REGION Network 11: Extrusora 11
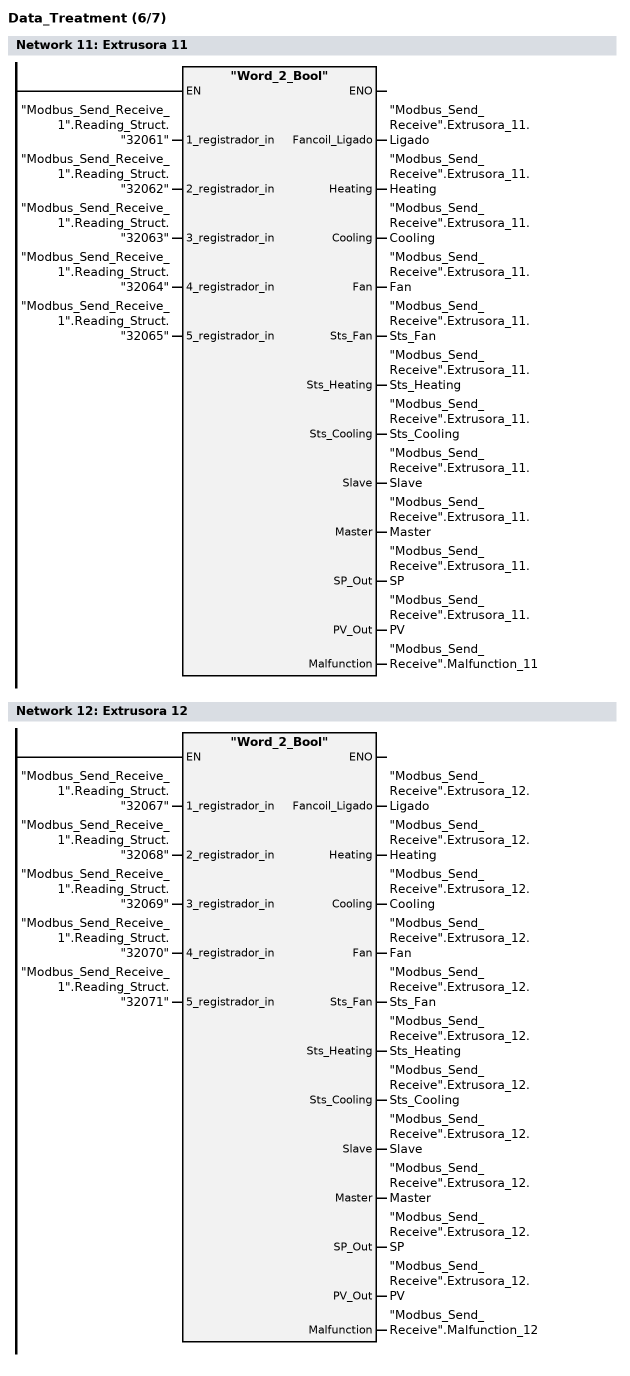
   RUNG wire#powerrail
      "Word_2_Bool"("1_registrador_in" := "Modbus_Send_Receive_1".Reading_Struct."32061", "2_registrador_in" := "Modbus_Send_Receive_1".Reading_Struct."32062", "3_registrador_in" := "Modbus_Send_Receive_1".Reading_Struct."32063", "4_registrador_in" := "Modbus_Send_Receive_1".Reading_Struct."32064", "5_registrador_in" := "Modbus_Send_Receive_1".Reading_Struct."32065", Fancoil_Ligado => "Modbus_Send_Receive".Extrusora_11.Ligado, Heating => "Modbus_Send_Receive".Extrusora_11.Heating, Cooling => "Modbus_Send_Receive".Extrusora_11.Cooling, Fan => "Modbus_Send_Receive".Extrusora_11.Fan, Sts_Fan => "Modbus_Send_Receive".Extrusora_11.Sts_Fan, Sts_Heating => "Modbus_Send_Receive".Extrusora_11.Sts_Heating, Sts_Cooling => "Modbus_Send_Receive".Extrusora_11.Sts_Cooling, Slave => "Modbus_Send_Receive".Extrusora_11.Slave, Master => "Modbus_Send_Receive".Extrusora_11.Master, SP_Out => "Modbus_Send_Receive".Extrusora_11.SP, PV_Out => "Modbus_Send_Receive".Extrusora_11.PV, Malfunction => "Modbus_Send_Receive".Malfunction_11)
   END_RUNG
   // the same network as SCL:
   "Word_2_Bool"("1_registrador_in" := "Modbus_Send_Receive_1".Reading_Struct."32061",
                 "2_registrador_in" := "Modbus_Send_Receive_1".Reading_Struct."32062",
                 "3_registrador_in" := "Modbus_Send_Receive_1".Reading_Struct."32063",
                 "4_registrador_in" := "Modbus_Send_Receive_1".Reading_Struct."32064",
                 "5_registrador_in" := "Modbus_Send_Receive_1".Reading_Struct."32065",
                 Fancoil_Ligado => "Modbus_Send_Receive".Extrusora_11.Ligado,
                 Heating => "Modbus_Send_Receive".Extrusora_11.Heating,
                 Cooling => "Modbus_Send_Receive".Extrusora_11.Cooling,
                 Fan => "Modbus_Send_Receive".Extrusora_11.Fan,
                 Sts_Fan => "Modbus_Send_Receive".Extrusora_11.Sts_Fan,
                 Sts_Heating => "Modbus_Send_Receive".Extrusora_11.Sts_Heating,
                 Sts_Cooling => "Modbus_Send_Receive".Extrusora_11.Sts_Cooling,
                 Slave => "Modbus_Send_Receive".Extrusora_11.Slave,
                 Master => "Modbus_Send_Receive".Extrusora_11.Master,
                 SP_Out => "Modbus_Send_Receive".Extrusora_11.SP,
                 PV_Out => "Modbus_Send_Receive".Extrusora_11.PV,
                 Malfunction => "Modbus_Send_Receive".Malfunction_11);
END_REGION

REGION Network 12: Extrusora 12
   RUNG wire#powerrail
      "Word_2_Bool"("1_registrador_in" := "Modbus_Send_Receive_1".Reading_Struct."32067", "2_registrador_in" := "Modbus_Send_Receive_1".Reading_Struct."32068", "3_registrador_in" := "Modbus_Send_Receive_1".Reading_Struct."32069", "4_registrador_in" := "Modbus_Send_Receive_1".Reading_Struct."32070", "5_registrador_in" := "Modbus_Send_Receive_1".Reading_Struct."32071", Fancoil_Ligado => "Modbus_Send_Receive".Extrusora_12.Ligado, Heating => "Modbus_Send_Receive".Extrusora_12.Heating, Cooling => "Modbus_Send_Receive".Extrusora_12.Cooling, Fan => "Modbus_Send_Receive".Extrusora_12.Fan, Sts_Fan => "Modbus_Send_Receive".Extrusora_12.Sts_Fan, Sts_Heating => "Modbus_Send_Receive".Extrusora_12.Sts_Heating, Sts_Cooling => "Modbus_Send_Receive".Extrusora_12.Sts_Cooling, Slave => "Modbus_Send_Receive".Extrusora_12.Slave, Master => "Modbus_Send_Receive".Extrusora_12.Master, SP_Out => "Modbus_Send_Receive".Extrusora_12.SP, PV_Out => "Modbus_Send_Receive".Extrusora_12.PV, Malfunction => "Modbus_Send_Receive".Malfunction_12)
   END_RUNG
   // the same network as SCL:
   "Word_2_Bool"("1_registrador_in" := "Modbus_Send_Receive_1".Reading_Struct."32067",
                 "2_registrador_in" := "Modbus_Send_Receive_1".Reading_Struct."32068",
                 "3_registrador_in" := "Modbus_Send_Receive_1".Reading_Struct."32069",
                 "4_registrador_in" := "Modbus_Send_Receive_1".Reading_Struct."32070",
                 "5_registrador_in" := "Modbus_Send_Receive_1".Reading_Struct."32071",
                 Fancoil_Ligado => "Modbus_Send_Receive".Extrusora_12.Ligado,
                 Heating => "Modbus_Send_Receive".Extrusora_12.Heating,
                 Cooling => "Modbus_Send_Receive".Extrusora_12.Cooling,
                 Fan => "Modbus_Send_Receive".Extrusora_12.Fan,
                 Sts_Fan => "Modbus_Send_Receive".Extrusora_12.Sts_Fan,
                 Sts_Heating => "Modbus_Send_Receive".Extrusora_12.Sts_Heating,
                 Sts_Cooling => "Modbus_Send_Receive".Extrusora_12.Sts_Cooling,
                 Slave => "Modbus_Send_Receive".Extrusora_12.Slave,
                 Master => "Modbus_Send_Receive".Extrusora_12.Master,
                 SP_Out => "Modbus_Send_Receive".Extrusora_12.SP,
                 PV_Out => "Modbus_Send_Receive".Extrusora_12.PV,
                 Malfunction => "Modbus_Send_Receive".Malfunction_12);
END_REGION

REGION Network 13: Extrusora 13
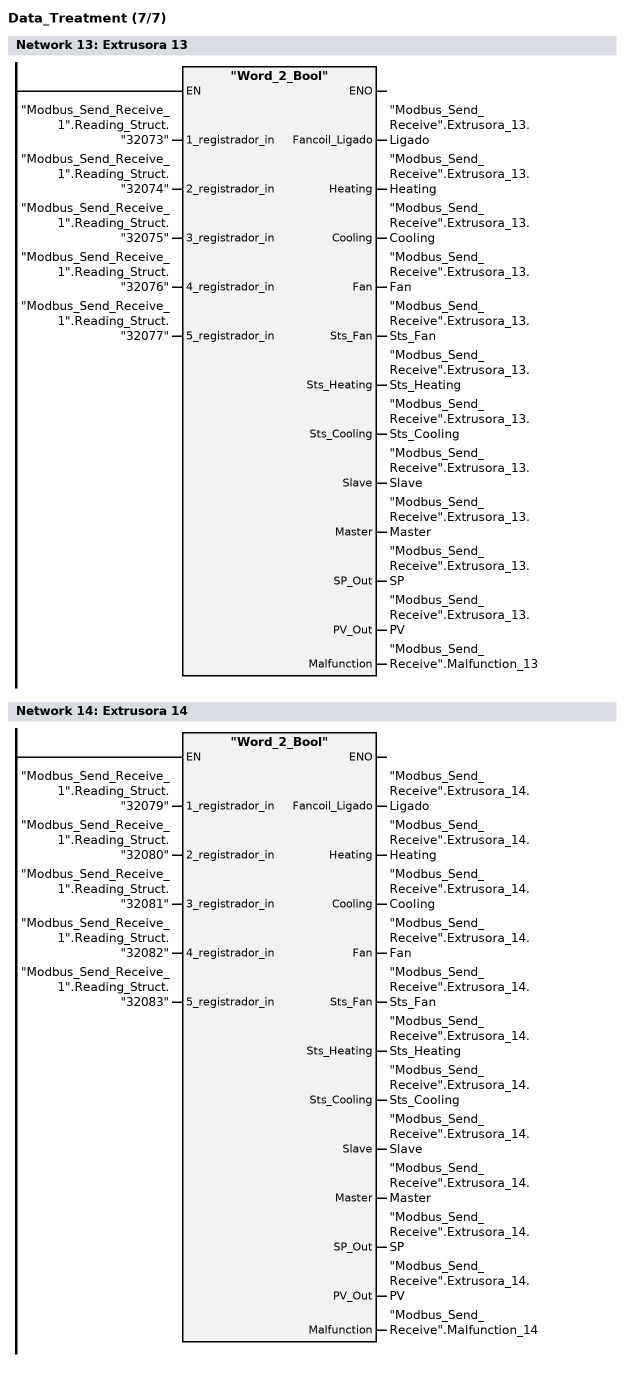
   RUNG wire#powerrail
      "Word_2_Bool"("1_registrador_in" := "Modbus_Send_Receive_1".Reading_Struct."32073", "2_registrador_in" := "Modbus_Send_Receive_1".Reading_Struct."32074", "3_registrador_in" := "Modbus_Send_Receive_1".Reading_Struct."32075", "4_registrador_in" := "Modbus_Send_Receive_1".Reading_Struct."32076", "5_registrador_in" := "Modbus_Send_Receive_1".Reading_Struct."32077", Fancoil_Ligado => "Modbus_Send_Receive".Extrusora_13.Ligado, Heating => "Modbus_Send_Receive".Extrusora_13.Heating, Cooling => "Modbus_Send_Receive".Extrusora_13.Cooling, Fan => "Modbus_Send_Receive".Extrusora_13.Fan, Sts_Fan => "Modbus_Send_Receive".Extrusora_13.Sts_Fan, Sts_Heating => "Modbus_Send_Receive".Extrusora_13.Sts_Heating, Sts_Cooling => "Modbus_Send_Receive".Extrusora_13.Sts_Cooling, Slave => "Modbus_Send_Receive".Extrusora_13.Slave, Master => "Modbus_Send_Receive".Extrusora_13.Master, SP_Out => "Modbus_Send_Receive".Extrusora_13.SP, PV_Out => "Modbus_Send_Receive".Extrusora_13.PV, Malfunction => "Modbus_Send_Receive".Malfunction_13)
   END_RUNG
   // the same network as SCL:
   "Word_2_Bool"("1_registrador_in" := "Modbus_Send_Receive_1".Reading_Struct."32073",
                 "2_registrador_in" := "Modbus_Send_Receive_1".Reading_Struct."32074",
                 "3_registrador_in" := "Modbus_Send_Receive_1".Reading_Struct."32075",
                 "4_registrador_in" := "Modbus_Send_Receive_1".Reading_Struct."32076",
                 "5_registrador_in" := "Modbus_Send_Receive_1".Reading_Struct."32077",
                 Fancoil_Ligado => "Modbus_Send_Receive".Extrusora_13.Ligado,
                 Heating => "Modbus_Send_Receive".Extrusora_13.Heating,
                 Cooling => "Modbus_Send_Receive".Extrusora_13.Cooling,
                 Fan => "Modbus_Send_Receive".Extrusora_13.Fan,
                 Sts_Fan => "Modbus_Send_Receive".Extrusora_13.Sts_Fan,
                 Sts_Heating => "Modbus_Send_Receive".Extrusora_13.Sts_Heating,
                 Sts_Cooling => "Modbus_Send_Receive".Extrusora_13.Sts_Cooling,
                 Slave => "Modbus_Send_Receive".Extrusora_13.Slave,
                 Master => "Modbus_Send_Receive".Extrusora_13.Master,
                 SP_Out => "Modbus_Send_Receive".Extrusora_13.SP,
                 PV_Out => "Modbus_Send_Receive".Extrusora_13.PV,
                 Malfunction => "Modbus_Send_Receive".Malfunction_13);
END_REGION

REGION Network 14: Extrusora 14
   RUNG wire#powerrail
      "Word_2_Bool"("1_registrador_in" := "Modbus_Send_Receive_1".Reading_Struct."32079", "2_registrador_in" := "Modbus_Send_Receive_1".Reading_Struct."32080", "3_registrador_in" := "Modbus_Send_Receive_1".Reading_Struct."32081", "4_registrador_in" := "Modbus_Send_Receive_1".Reading_Struct."32082", "5_registrador_in" := "Modbus_Send_Receive_1".Reading_Struct."32083", Fancoil_Ligado => "Modbus_Send_Receive".Extrusora_14.Ligado, Heating => "Modbus_Send_Receive".Extrusora_14.Heating, Cooling => "Modbus_Send_Receive".Extrusora_14.Cooling, Fan => "Modbus_Send_Receive".Extrusora_14.Fan, Sts_Fan => "Modbus_Send_Receive".Extrusora_14.Sts_Fan, Sts_Heating => "Modbus_Send_Receive".Extrusora_14.Sts_Heating, Sts_Cooling => "Modbus_Send_Receive".Extrusora_14.Sts_Cooling, Slave => "Modbus_Send_Receive".Extrusora_14.Slave, Master => "Modbus_Send_Receive".Extrusora_14.Master, SP_Out => "Modbus_Send_Receive".Extrusora_14.SP, PV_Out => "Modbus_Send_Receive".Extrusora_14.PV, Malfunction => "Modbus_Send_Receive".Malfunction_14)
   END_RUNG
   // the same network as SCL:
   "Word_2_Bool"("1_registrador_in" := "Modbus_Send_Receive_1".Reading_Struct."32079",
                 "2_registrador_in" := "Modbus_Send_Receive_1".Reading_Struct."32080",
                 "3_registrador_in" := "Modbus_Send_Receive_1".Reading_Struct."32081",
                 "4_registrador_in" := "Modbus_Send_Receive_1".Reading_Struct."32082",
                 "5_registrador_in" := "Modbus_Send_Receive_1".Reading_Struct."32083",
                 Fancoil_Ligado => "Modbus_Send_Receive".Extrusora_14.Ligado,
                 Heating => "Modbus_Send_Receive".Extrusora_14.Heating,
                 Cooling => "Modbus_Send_Receive".Extrusora_14.Cooling,
                 Fan => "Modbus_Send_Receive".Extrusora_14.Fan,
                 Sts_Fan => "Modbus_Send_Receive".Extrusora_14.Sts_Fan,
                 Sts_Heating => "Modbus_Send_Receive".Extrusora_14.Sts_Heating,
                 Sts_Cooling => "Modbus_Send_Receive".Extrusora_14.Sts_Cooling,
                 Slave => "Modbus_Send_Receive".Extrusora_14.Slave,
                 Master => "Modbus_Send_Receive".Extrusora_14.Master,
                 SP_Out => "Modbus_Send_Receive".Extrusora_14.SP,
                 PV_Out => "Modbus_Send_Receive".Extrusora_14.PV,
                 Malfunction => "Modbus_Send_Receive".Malfunction_14);
END_REGION
END_FUNCTION

FUNCTION "Word_2_Bool" : Void   // FC1, LAD
{ S7_Optimized_Access := 'TRUE' }
VERSION : 0.1
// stored: AutoNumber true, IsIECCheckEnabled false, SetENOAutomatically false, UDAEnableTagReadback false
   VAR_INPUT
      "1_registrador_in" : Word;
      "2_registrador_in" : Word;
      "3_registrador_in" : Word;
      "4_registrador_in" : Word;
      "5_registrador_in" : Word;
   END_VAR
   VAR_OUTPUT
      Fancoil_Ligado : Bool;
      Heating : Bool;
      Cooling : Bool;
      Fan : Bool;
      Sts_Fan : Bool;
      Sts_Heating : Bool;
      Sts_Cooling : Bool;
      Slave : Bool;
      Master : Bool;
      SP_Out : Real;
      PV_Out : Real;
      Malfunction : Bool;
   END_VAR
   VAR_TEMP
      Aux_1 : Word;
      Aux_2 : Word;
      Aux_3 : Word;
      Aux_4 : Word;
      Temp_Real_Word_1 : Real;
      Temp_Real_Word_2 : Real;
   END_VAR
BEGIN

REGION Network 1: Verifica se esta ligado ou desligado
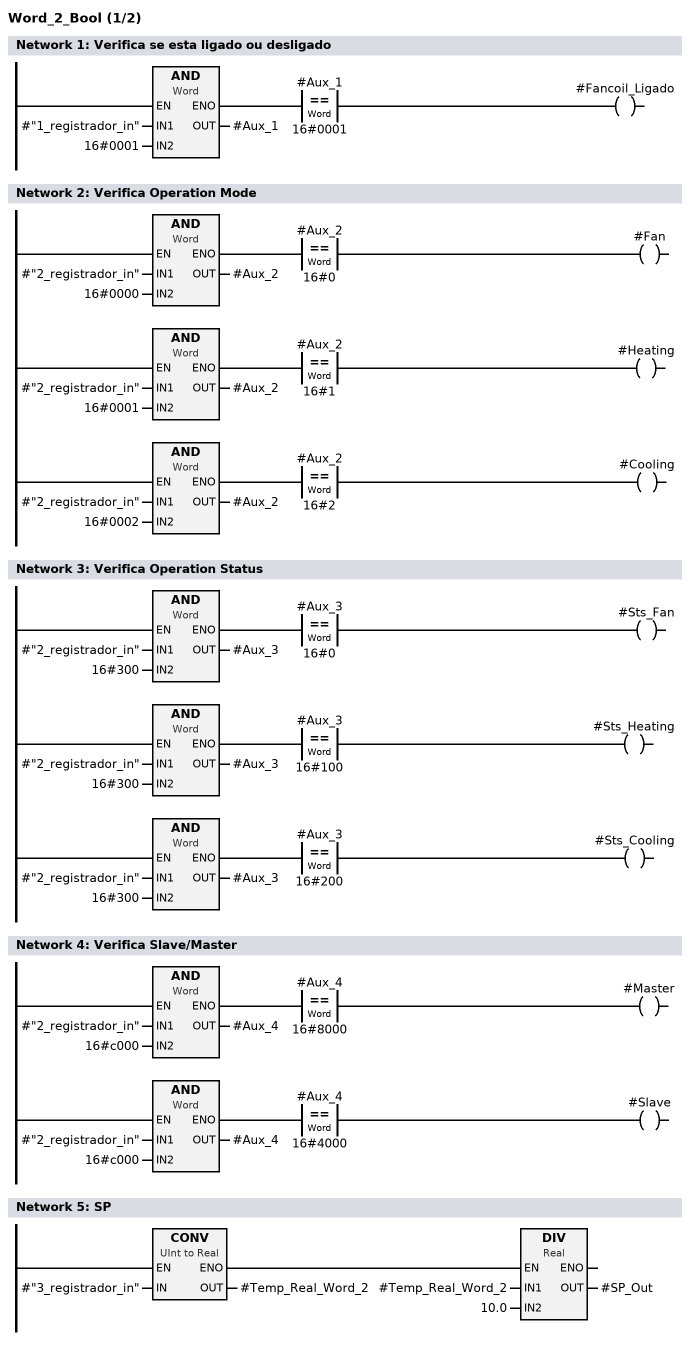
   RUNG wire#powerrail
      { S7_Templates := "SrcType := Word" } And(in1 := #"1_registrador_in", in2 := 16#0001, out => #Aux_1)
      { S7_Templates := "SrcType := Word" } EQ_Contact(in1 := #Aux_1, in2 := 16#0001)
      Coil( #Fancoil_Ligado )
   END_RUNG
   // the same network as SCL:
   #Aux_1 := #"1_registrador_in" AND 16#0001;
   #Fancoil_Ligado := #Aux_1 = 16#0001;
END_REGION

REGION Network 2: Verifica Operation Mode
   RUNG wire#powerrail
      { S7_Templates := "SrcType := Word" } And(in1 := #"2_registrador_in", in2 := 16#0000, out => #Aux_2)
      { S7_Templates := "SrcType := Word" } EQ_Contact(in1 := #Aux_2, in2 := 16#0)
      Coil( #Fan )
   END_RUNG
   RUNG wire#powerrail
      { S7_Templates := "SrcType := Word" } And(in1 := #"2_registrador_in", in2 := 16#0001, out => #Aux_2)
      { S7_Templates := "SrcType := Word" } EQ_Contact(in1 := #Aux_2, in2 := 16#1)
      Coil( #Heating )
   END_RUNG
   RUNG wire#powerrail
      { S7_Templates := "SrcType := Word" } And(in1 := #"2_registrador_in", in2 := 16#0002, out => #Aux_2)
      { S7_Templates := "SrcType := Word" } EQ_Contact(in1 := #Aux_2, in2 := 16#2)
      Coil( #Cooling )
   END_RUNG
   // the same network as SCL:
   #Aux_2 := #"2_registrador_in" AND 16#0000;
   #Fan := #Aux_2 = 16#0;
   #Aux_2 := #"2_registrador_in" AND 16#0001;
   #Heating := #Aux_2 = 16#1;
   #Aux_2 := #"2_registrador_in" AND 16#0002;
   #Cooling := #Aux_2 = 16#2;
END_REGION

REGION Network 3: Verifica Operation Status
   RUNG wire#powerrail
      { S7_Templates := "SrcType := Word" } And(in1 := #"2_registrador_in", in2 := 16#300, out => #Aux_3)
      { S7_Templates := "SrcType := Word" } EQ_Contact(in1 := #Aux_3, in2 := 16#0)
      Coil( #Sts_Fan )
   END_RUNG
   RUNG wire#powerrail
      { S7_Templates := "SrcType := Word" } And(in1 := #"2_registrador_in", in2 := 16#300, out => #Aux_3)
      { S7_Templates := "SrcType := Word" } EQ_Contact(in1 := #Aux_3, in2 := 16#100)
      Coil( #Sts_Heating )
   END_RUNG
   RUNG wire#powerrail
      { S7_Templates := "SrcType := Word" } And(in1 := #"2_registrador_in", in2 := 16#300, out => #Aux_3)
      { S7_Templates := "SrcType := Word" } EQ_Contact(in1 := #Aux_3, in2 := 16#200)
      Coil( #Sts_Cooling )
   END_RUNG
   // the same network as SCL:
   #Aux_3 := #"2_registrador_in" AND 16#300;
   #Sts_Fan := #Aux_3 = 16#0;
   #Aux_3 := #"2_registrador_in" AND 16#300;
   #Sts_Heating := #Aux_3 = 16#100;
   #Aux_3 := #"2_registrador_in" AND 16#300;
   #Sts_Cooling := #Aux_3 = 16#200;
END_REGION

REGION Network 4: Verifica Slave/Master
   RUNG wire#powerrail
      { S7_Templates := "SrcType := Word" } And(in1 := #"2_registrador_in", in2 := 16#c000, out => #Aux_4)
      { S7_Templates := "SrcType := Word" } EQ_Contact(in1 := #Aux_4, in2 := 16#8000)
      Coil( #Master )
   END_RUNG
   RUNG wire#powerrail
      { S7_Templates := "SrcType := Word" } And(in1 := #"2_registrador_in", in2 := 16#c000, out => #Aux_4)
      { S7_Templates := "SrcType := Word" } EQ_Contact(in1 := #Aux_4, in2 := 16#4000)
      Coil( #Slave )
   END_RUNG
   // the same network as SCL:
   #Aux_4 := #"2_registrador_in" AND 16#c000;
   #Master := #Aux_4 = 16#8000;
   #Aux_4 := #"2_registrador_in" AND 16#c000;
   #Slave := #Aux_4 = 16#4000;
END_REGION

REGION Network 5: SP
   RUNG wire#powerrail
      { S7_Templates := "[SrcType := UInt, DestType := Real]" } Convert(in := #"3_registrador_in", out => #Temp_Real_Word_2)
      { S7_Templates := "SrcType := Real" } Div(in1 := #Temp_Real_Word_2, in2 := 10.0, out => #SP_Out)
   END_RUNG
   // the same network as SCL:
   #Temp_Real_Word_2 := UINT_TO_REAL(#"3_registrador_in");
   #SP_Out := #Temp_Real_Word_2 / 10.0;
END_REGION

REGION Network 6: PV
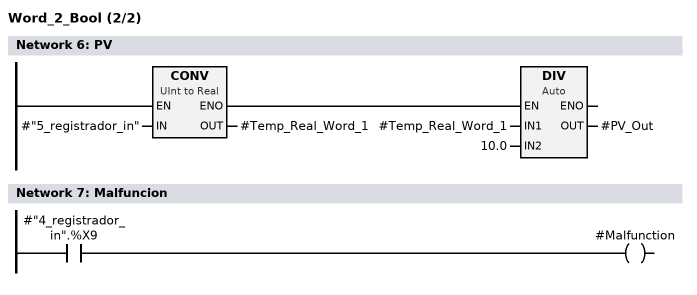
   RUNG wire#powerrail
      { S7_Templates := "[SrcType := UInt, DestType := Real]" } Convert(in := #"5_registrador_in", out => #Temp_Real_Word_1)
      Div(in1 := #Temp_Real_Word_1, in2 := 10.0, out => #PV_Out)
   END_RUNG
   // the same network as SCL:
   #Temp_Real_Word_1 := UINT_TO_REAL(#"5_registrador_in");
   #PV_Out := #Temp_Real_Word_1 / 10.0;
END_REGION

REGION Network 7: Malfuncion
   RUNG wire#powerrail
      Contact( #"4_registrador_in".%X9 )
      Coil( #Malfunction )
   END_RUNG
   // the same network as SCL:
   #Malfunction := #"4_registrador_in".%X9;
END_REGION
END_FUNCTION

DATA_BLOCK "MB_COMM_Setup_dB"   // DB9
VERSION : 0.1
// stored: AutoNumber true, DBAccessibleFromOPCUA true, InstanceOfName MB_Comm_Setup, InstanceOfType FB
"MB_Comm_Setup"
BEGIN
END_DATA_BLOCK

DATA_BLOCK "IEC_Counter_0_DB"   // DB4
{ S7_Optimized_Access := 'TRUE' }
// stored: AutoNumber true, DBAccessibleFromOPCUA true, InstanceOfName IEC_COUNTER, OfSystemLibElement IEC_COUNTER, OfSystemLibVersion 1.0
"IEC_COUNTER"
   // VAR RETAIN
   //    CU : Bool;
   //    CD : Bool;
   //    R : Bool;
   //    LD : Bool;
   //    QU : Bool;
   //    QD : Bool;
   //    PV : Int;
   //    CV : Int;
   // END_VAR
BEGIN
END_DATA_BLOCK

DATA_BLOCK "IEC_Counter_0_DB_1"   // DB6
{ S7_Optimized_Access := 'TRUE' }
// stored: AutoNumber true, DBAccessibleFromOPCUA true, InstanceOfName IEC_COUNTER, OfSystemLibElement IEC_COUNTER, OfSystemLibVersion 1.0
"IEC_COUNTER"
   // VAR RETAIN
   //    CU : Bool;
   //    CD : Bool;
   //    R : Bool;
   //    LD : Bool;
   //    QU : Bool;
   //    QD : Bool;
   //    PV : Int;
   //    CV : Int;
   // END_VAR
BEGIN
END_DATA_BLOCK

DATA_BLOCK "IEC_Counter_0_DB_2"   // DB7
{ S7_Optimized_Access := 'TRUE' }
// stored: AutoNumber true, DBAccessibleFromOPCUA true, InstanceOfName IEC_COUNTER, OfSystemLibElement IEC_COUNTER, OfSystemLibVersion 1.0
"IEC_COUNTER"
   // VAR RETAIN
   //    CU : Bool;
   //    CD : Bool;
   //    R : Bool;
   //    LD : Bool;
   //    QU : Bool;
   //    QD : Bool;
   //    PV : Int;
   //    CV : Int;
   // END_VAR
BEGIN
END_DATA_BLOCK

DATA_BLOCK "IEC_Timer_0_DB"   // DB8
{ S7_Optimized_Access := 'TRUE' }
// stored: AutoNumber true, DBAccessibleFromOPCUA true, InstanceOfName IEC_TIMER, OfSystemLibElement IEC_TIMER, OfSystemLibVersion 1.0
"IEC_TIMER"
   // VAR
   //    PT : Time;
   //    ET { ExternalWritable := 'False'} : Time;
   //    IN : Bool;
   //    Q { ExternalWritable := 'False'} : Bool;
   // END_VAR
BEGIN
END_DATA_BLOCK

DATA_BLOCK "IEC_Timer_0_DB_1"   // DB11
{ S7_Optimized_Access := 'TRUE' }
// stored: AutoNumber true, DBAccessibleFromOPCUA true, InstanceOfName IEC_TIMER, OfSystemLibElement IEC_TIMER, OfSystemLibVersion 1.0
"IEC_TIMER"
   // VAR
   //    PT : Time;
   //    ET { ExternalWritable := 'False'} : Time;
   //    IN : Bool;
   //    Q { ExternalWritable := 'False'} : Bool;
   // END_VAR
BEGIN
END_DATA_BLOCK

DATA_BLOCK "Modbus_Comm_Load_DB"   // DB2
// stored: AutoNumber true, DBAccessibleFromOPCUA true, InstanceOfName Modbus_Comm_Load, OfSystemLibElement Modbus_Comm_Load, OfSystemLibVersion 3.1
"Modbus_Comm_Load"
   // VAR_INPUT
   //    REQ : Bool;
   //    PORT : PORT;
   //    BAUD : UDInt;
   //    PARITY : UInt;
   //    FLOW_CTRL : UInt;
   //    RTS_ON_DLY : UInt;
   //    RTS_OFF_DLY : UInt;
   //    RESP_TO : UInt;
   // END_VAR
   // VAR_OUTPUT
   //    DONE : Bool;
   //    ERROR : Bool;
   //    STATUS : Word;
   // END_VAR
   // VAR_IN_OUT
   //    MB_DB : P2P_MB_BASE;
   // END_VAR
   // VAR
   //    ICHAR_GAP : Word;
   //    RETRIES : Word;
   //    MODE : USInt;
   //    LINE_PRE : USInt;
   //    BRK_DET : USInt;
   //    EN_DIAG_ALARM : Bool;
   //    STOP_BITS : USInt;
   //    EN_SUPPLY_VOLT : Bool;
   //    b_e_REQ : Bool;
   //    y_state : SInt;
   //    Send_Config { S7_SetPoint := 'True'} : Send_Config;
   //    Receive_Config { S7_SetPoint := 'True'} : Receive_Config;
   //    Receive_Conditions { S7_SetPoint := 'True'} : Receive_Conditions;
   //    WRREC { S7_SetPoint := 'True'} : WRREC;
   //    RDREC { S7_SetPoint := 'True'} : RDREC;
   //    port_w_record { ExternalVisible := 'False'; S7_SetPoint := 'True'} : P2P_MB_PortData;
   //    err_record { ExternalVisible := 'False'; S7_SetPoint := 'True'} : P2P_RdEstat;
   //    ftrs_w_record { ExternalVisible := 'False'; S7_SetPoint := 'True'} : P2P_FeaturesData;
   //    wlen : UInt;
   // END_VAR
BEGIN
END_DATA_BLOCK

DATA_BLOCK "Modbus_Master_DB"   // DB3
// stored: AutoNumber true, DBAccessibleFromOPCUA true, InstanceOfName Modbus_Master, OfSystemLibElement Modbus_Master, OfSystemLibVersion 3.3
"Modbus_Master"
   // VAR_INPUT
   //    REQ : Bool;
   //    MB_ADDR : UInt;
   //    MODE : USInt;
   //    DATA_ADDR : UDInt;
   //    DATA_LEN : UInt;
   // END_VAR
   // VAR_OUTPUT
   //    DONE : Bool;
   //    BUSY : Bool;
   //    ERROR : Bool;
   //    STATUS : Word;
   // END_VAR
   // VAR_IN_OUT
   //    DATA_PTR : Variant;
   // END_VAR
   // VAR
   //    MB_State : SInt;
   //    Blocked_Proc_Timeout : Real;
   //    Extended_Addressing : Bool;
   //    Compatibility_Mode : Bool;
   //    MB_DB { S7_SetPoint := 'True'} : P2P_MB_BASE;
   //    Send_P2P { S7_SetPoint := 'True'} : Send_P2P;
   //    Receive_P2P { S7_SetPoint := 'True'} : Receive_P2P;
   //    Receive_Reset { S7_SetPoint := 'True'} : Receive_Reset;
   //    S_PORT : Word;
   //    S_RESP_TO : Word;
   //    S_ICHAR_GAP : Word;
   //    S_RETRIES : Word;
   //    S_MB_ADDR : UInt;
   //    S_MODE : USInt;
   //    S_DATA_ADDR : UDInt;
   //    S_DATA_LEN : UInt;
   //    w_retries : Word;
   //    y_SlaveAddrHi : Byte;
   //    y_SlaveAddrLo : Byte;
   //    StartAddress : Word;
   //    Value : Word;
   //    y_FCode : Byte;
   //    INTERNAL_CDATA : Array[1..257] of Byte;
   //    mb_timer { S7_SetPoint := 'True'} : TON_TIME;
   //    TimeElapsed : Bool;
   // END_VAR
BEGIN
END_DATA_BLOCK
